% RSLogix 500 project PROC1_ANALOG_IO_BAK000.RSS, saved by version 8.30.00.16 %
PROJECT "PROC1"    % processor: Bul.1763 MicroLogix 1100 Series B %

PROGRAM FILES
  LAD 2 "MAIN"  1 rungs
  LAD 3 "ANALOG IO"  2 rungs

DATA FILES
  O0 OUTPUT  6 elements
  I1 INPUT  12 elements
  S2 STATUS  66 elements
  B3 BINARY  1 elements
  T4 TIMER  1 elements
  C5 COUNTER  1 elements
  R6 CONTROL  1 elements
  N7 INTEGER  1 elements
  F8 FLOAT  1 elements

LADDER 3 "ANALOG IO"
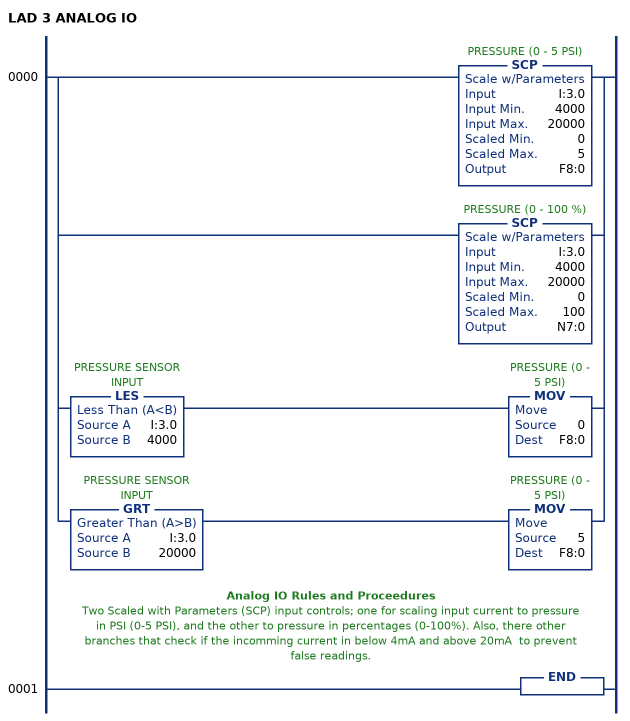
% Rung: 0 %  % edit flag set %
SOR BST SCP I:3.0 4000 20000 0 5 F8:0 NXB SCP I:3.0 4000 20000 0 100 N7:0 NXB LES I:3.0 4000 MOV 0 F8:0 NXB GRT I:3.0 20000 MOV 5 F8:0 BND EOR
%   I:3.0  "PRESSURE SENSOR INPUT" %
%   F8:0  "PRESSURE (0 - 5 PSI)" %
%   N7:0  "PRESSURE (0 - 100 %)" %
% Rung: 1 %
% TITLE: Analog IO Rules and Proceedures %
% Two Scaled with Parameters (SCP) input controls; one for scaling input current to pressure in PSI (0-5 PSI), and the other to pressure in percentages (0-100%). Also, there other branches that check if the incomming current in below 4mA and above 20mA  to prevent false readings. %
SOR END EOR
